FUNCTION FC_GetMaxValue : REAL
VAR_INPUT
END_VAR
VAR
	iCurrentPos: INT;
END_VAR
VAR_IN_OUT
	MaxValue: ARRAY[0..100] OF REAL;
END_VAR

MaxValue[0] := 0;

FOR iCurrentPos := 1 TO 100 BY 1 DO
	IF MaxValue[iCurrentPos] > MaxValue[0] THEN
		MaxValue[0] := MaxValue[iCurrentPos];
	END_IF
END_FOR

FC_GetMaxValue := MaxValue[0];

END_FUNCTION

(* stored: Version 1.1.0.1
   POU FC_GetMaxValue: Id {e134bd17-db76-4c1d-9f5a-3d4721a1e675}, SpecialFunc None *)
